Staubli VAL3: encodePoint.pgx

program encodePoint(point& value, num& buffer[])
  local num elements[6]
begin
  elements[0] = value.trsf.x
  elements[1] = value.trsf.y
  elements[2] = value.trsf.z
  elements[3] = value.trsf.rx
  elements[4] = value.trsf.ry
  elements[5] = value.trsf.rz

  toBinary(elements, 6, "4.0b", buffer)
end
